//==================================================================================================
//							Beckhoff Automation Poland
//									11.04.2018
//	This object shall provide the text id of the last DiagMessage of type error, which occurred in this axis.
//  v1.0	|| TC v 3.1.4022.16		|| - pierwsza wersja
//==================================================================================================
FUNCTION_BLOCK FB_ReadChannelErrorCodeAX8000
VAR_INPUT
	bExecute 						: BOOL;
	stDriveRef						: ST_DriveRef;						// 
END_VAR
VAR_OUTPUT
	bBusy							: BOOL;
	bError							: BOOL; 							// General error: parameter or CoE read.
	iAdsErrId						: UINT;								// Forwarded output FB_CoERead_ByDriveRef
	iCANopenErrId					: UINT;								// Forwarded output FB_CoERead_ByDriveRef
	uiChannelErrorCode				: UINT;								// 603F Error code	0x603F (Ch A)/ 0x683F (Ch B) 	UINT16
	{attribute 'displaymode':='hex'}
	uiChannelErrorCodeHex			: UINT;								// 603F Error code	0x603F (Ch A)/ 0x683F (Ch B) 	UINT16
END_VAR
VAR
	fbCoERead						: FB_CoERead_ByDriveRef;			// FB for read CoE parameters
END_VAR

fbCoERead(	stDriveRef					:= stDriveRef,
			nIndex						:= 16#603F + (stDriveRef.nDriveNo * 16#800),
			nSubIndex					:= 0,
			pDstBuf						:= ADR(uiChannelErrorCode),
			cbBufLen					:= SIZEOF(uiChannelErrorCode),
			bExecute					:= bExecute,
			bBusy						=> bBusy,
			bError						=> bError,
			iAdsErrId					=> iAdsErrId,
			iCANopenErrId				=> iCANopenErrId);

uiChannelErrorCodeHex					:= uiChannelErrorCode;

END_FUNCTION_BLOCK

(* stored: Version 1.1.0.1, ProductVersion 3.1.4026.13, FileIdentifier 1f062430a6b730cdc14bf215aa1c14d3625a45a4, FileSignature 6db5b1ff8f37507c81aa1669bf59ce22152581a885399bcd43fb8205350c3e99002c888349f51374dab5842cf3956b2bacc900e71cd7f160dfec1a3fb04a0f4a0dcbab83f63673f244360fa462c5e7f669c50af31900f5235f14030174f58abd675f15bb070b9bf4f4702a2be709a4e456424ab6b4fafccc9f302e0d99c6d67522fe1363853ce8098e44d0aa20ec50e5b14d5211fc343fc8fafd6304f36e732f6803fafbdaa0e60da2d32a792d1003c3ed1cb7cb5b50bda2958314c0440ae156e703a18bd387228f1926cc02e4e6b6cc57941c54cde77f4efefc5ea8f339758f88b9a264bc31ee6397b1a7ae5973cd3ae9022935dafd325c2e09d8c64e857746
   POU FB_ReadChannelErrorCodeAX8000: Id {449892ff-9e2a-4827-a4c7-2bb2ca0bb142}, SpecialFunc None *)
